(* Logix 5000 project; controller Google vendor 1 type 14 code 151 rev 31.11; software revision 31.00; part 2 of 6 *)

ADD_ON_INSTRUCTION Lift_Conv_Motor_Control   (* revision 1.0 *)
VAR_OUTPUT
   Motor_Data : SINT; {required}
END_VAR
VAR_INPUT
   Motor_FWD : BOOL; {required}
   Motor_REV : BOOL; {required}
   FWD_Speed : DINT; {required}
   REV_Speed : DINT; {required}
   Start_Delay : DINT; {required}
   Run_Permissive : DINT; {required}
END_VAR
VAR
   FWD_Delay : TIMER[4] := ([0].PRE := 500, [1].PRE := 500, [2].PRE := 500, [3].PRE := 500); {access None}
   REV_Delay : TIMER[4] := ([0].PRE := 500, [1].PRE := 500, [2].PRE := 500, [3].PRE := 500); {access None}
END_VAR

ROUTINE Logic   (* ladder *)
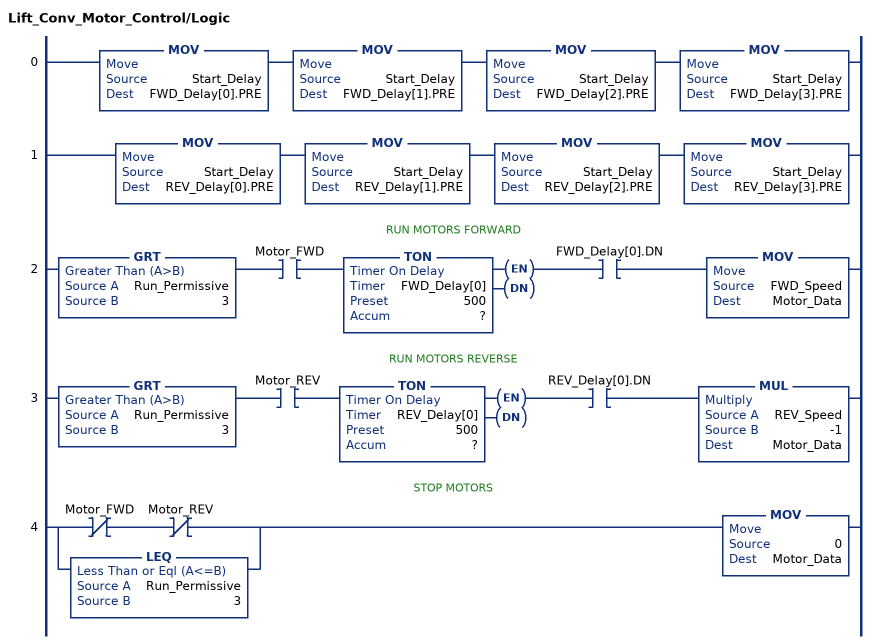
   0: MOV(Start_Delay,FWD_Delay[0].PRE)MOV(Start_Delay,FWD_Delay[1].PRE)MOV(Start_Delay,FWD_Delay[2].PRE)MOV(Start_Delay,FWD_Delay[3].PRE);
   1: MOV(Start_Delay,REV_Delay[0].PRE)MOV(Start_Delay,REV_Delay[1].PRE)MOV(Start_Delay,REV_Delay[2].PRE)MOV(Start_Delay,REV_Delay[3].PRE);
   // RUN MOTORS FORWARD
   2: GRT(Run_Permissive,3)XIC(Motor_FWD)TON(FWD_Delay[0],?,?)XIC(FWD_Delay[0].DN)MOV(FWD_Speed,Motor_Data);
   // RUN MOTORS REVERSE
   3: GRT(Run_Permissive,3)XIC(Motor_REV)TON(REV_Delay[0],?,?)XIC(REV_Delay[0].DN)MUL(REV_Speed,-1,Motor_Data);
   // STOP MOTORS
   4: [XIO(Motor_FWD) XIO(Motor_REV) ,LEQ(Run_Permissive,3) ]MOV(0,Motor_Data);
END_ROUTINE
END_ADD_ON_INSTRUCTION

ADD_ON_INSTRUCTION Lift_Conv_Sensor_Inputs   (* revision 1.0 *)
VAR_INPUT
   Data : SINT; {required}
END_VAR
VAR_OUTPUT
   Input_0 : BOOL; {access Read Only, required}
   Input_1 : BOOL; {access Read Only, required}
END_VAR

ROUTINE Logic   (* ladder *)
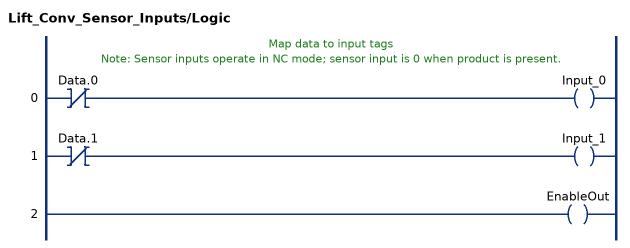
   // Map data to input tags
   // Note: Sensor inputs operate in NC mode; sensor input is 0 when product is present.
   0: XIO(Data.0)OTE(Input_0);
   1: XIO(Data.1)OTE(Input_1);
   2: OTE(EnableOut);
END_ROUTINE
END_ADD_ON_INSTRUCTION

ADD_ON_INSTRUCTION Lift_Zone_Data   (* revision 1.0 *)
VAR_IN_OUT
   Product_Name : STRING; {required}
   Product_Code : DINT; {required}
END_VAR
VAR_OUTPUT
   Occupied : BOOL; {access Read Only, visible}
END_VAR
VAR_INPUT
   Input_1 : BOOL; {required}
   Input_2 : BOOL; {required}
END_VAR
VAR_IN_OUT
   Upstream_ProdName : STRING; {required}
   Upstream_ProdCode : DINT; {required}
   Downstream_ProdName : STRING; {required}
   Downstream_ProdCode : DINT; {required}
END_VAR
VAR_INPUT
   FWD_Direction : BOOL; {required}
   REV_Direction : BOOL; {required}
END_VAR
VAR
   Blank_String : STRING; {access None}
   ONS : DINT; {access None}
   Occupied_Delay : TIMER := (PRE := 20); {access None}
   Unoccupied_Delay : TIMER := (PRE := 20); {access None}
END_VAR

ROUTINE Logic   (* ladder *)
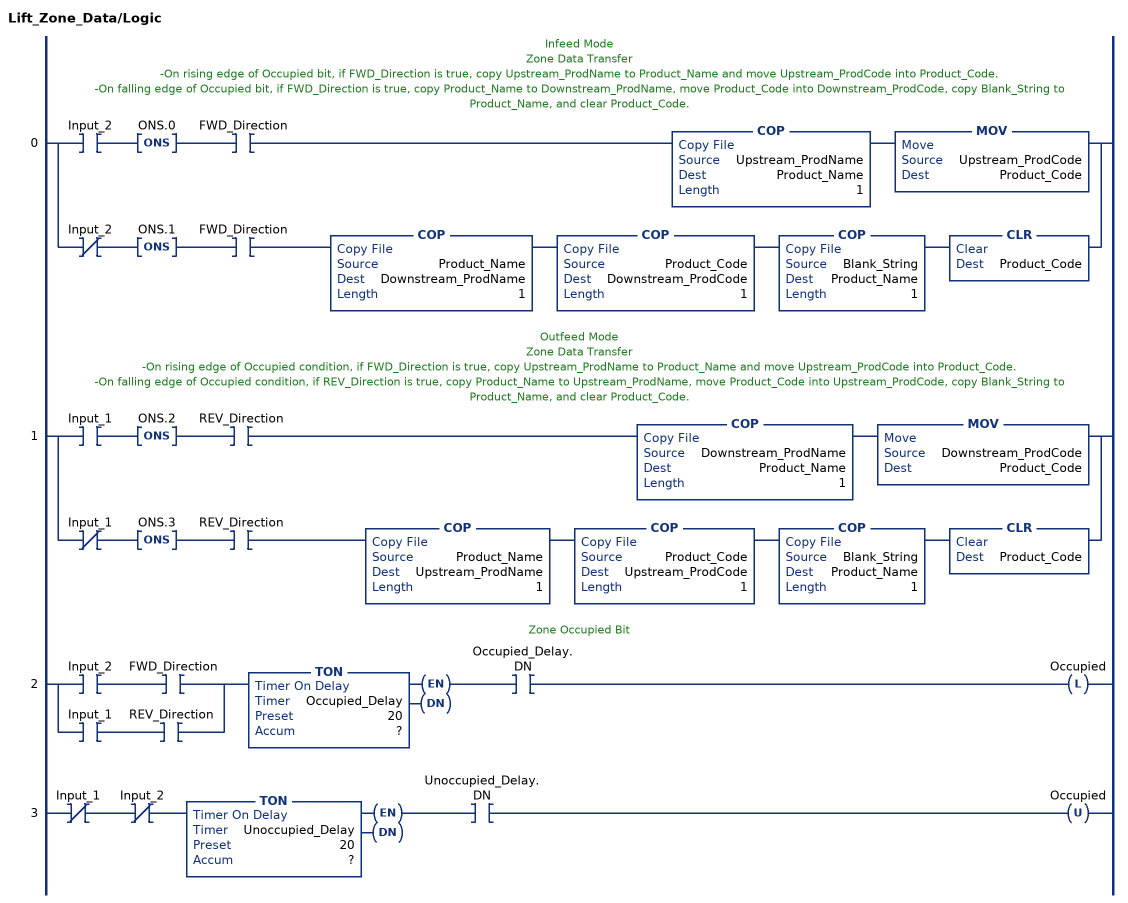
   // Infeed Mode
   // Zone Data Transfer
   // -On rising edge of Occupied bit, if FWD_Direction is true, copy Upstream_ProdName to Product_Name and move Upstream_ProdCode into Product_Code.
   // -On falling edge of Occupied bit, if FWD_Direction is true, copy Product_Name to Downstream_ProdName, move Product_Code into Downstream_ProdCode, copy Blank_String to Product_Name, and clear Product_Code.
   0: [XIC(Input_2) ONS(ONS.0) XIC(FWD_Direction) COP(Upstream_ProdName,Product_Name,1) MOV(Upstream_ProdCode,Product_Code) ,XIO(Input_2) ONS(ONS.1) XIC(FWD_Direction) COP(Product_Name,Downstream_ProdName,1) COP(Product_Code,Downstream_ProdCode,1) COP(Blank_String,Product_Name,1) CLR(Product_Code) ];
   // Outfeed Mode
   // Zone Data Transfer
   // -On rising edge of Occupied condition, if FWD_Direction is true, copy Upstream_ProdName to Product_Name and move Upstream_ProdCode into Product_Code.
   // -On falling edge of Occupied condition, if REV_Direction is true, copy Product_Name to Upstream_ProdName, move Product_Code into Upstream_ProdCode, copy Blank_String to Product_Name, and clear Product_Code.
   1: [XIC(Input_1) ONS(ONS.2) XIC(REV_Direction) COP(Downstream_ProdName,Product_Name,1) MOV(Downstream_ProdCode,Product_Code) ,XIO(Input_1) ONS(ONS.3) XIC(REV_Direction) COP(Product_Name,Upstream_ProdName,1) COP(Product_Code,Upstream_ProdCode,1) COP(Blank_String,Product_Name,1) CLR(Product_Code) ];
   // Zone Occupied Bit
   2: [XIC(Input_2) XIC(FWD_Direction) ,XIC(Input_1) XIC(REV_Direction) ]TON(Occupied_Delay,?,?)XIC(Occupied_Delay.DN)OTL(Occupied);
   3: XIO(Input_1)XIO(Input_2)TON(Unoccupied_Delay,?,?)XIC(Unoccupied_Delay.DN)OTU(Occupied);
END_ROUTINE
END_ADD_ON_INSTRUCTION

ADD_ON_INSTRUCTION Output_16_Bit   (* revision 1.0 *)
VAR_OUTPUT
   Output : BOOL; {access None}
   Data : INT; {required}
END_VAR
VAR_INPUT
   Output_0 : BOOL; {required}
   Output_1 : BOOL; {required}
   Output_2 : BOOL; {required}
   Output_3 : BOOL; {required}
   Output_4 : BOOL; {required}
   Output_5 : BOOL; {required}
   Output_6 : BOOL; {required}
   Output_7 : BOOL; {required}
   Output_8 : BOOL; {required}
   Output_9 : BOOL; {required}
   Output_10 : BOOL; {required}
   Output_11 : BOOL; {required}
   Output_12 : BOOL; {required}
   Output_13 : BOOL; {required}
   Output_14 : BOOL; {required}
   Output_15 : BOOL; {required}
   Test_Enable : BOOL; {required}
   Test_0 : BOOL; {required}
   Test_1 : BOOL; {required}
   Test_2 : BOOL; {required}
   Test_3 : BOOL; {required}
   Test_4 : BOOL; {required}
   Test_5 : BOOL; {required}
   Test_6 : BOOL; {required}
   Test_7 : BOOL; {required}
   Test_8 : BOOL; {required}
   Test_9 : BOOL; {required}
   Test_10 : BOOL; {required}
   Test_11 : BOOL; {required}
   Test_12 : BOOL; {required}
   Test_13 : BOOL; {required}
   Test_14 : BOOL; {required}
   Test_15 : BOOL; {required}
END_VAR
VAR
   ONS_Debounce : BOOL; {access None}
   Debounce_On_TMR : TIMER[16]; {access None}
   Debounce_Off_TMR : TIMER[16]; {access None}
END_VAR

ROUTINE Logic   (* ladder *)
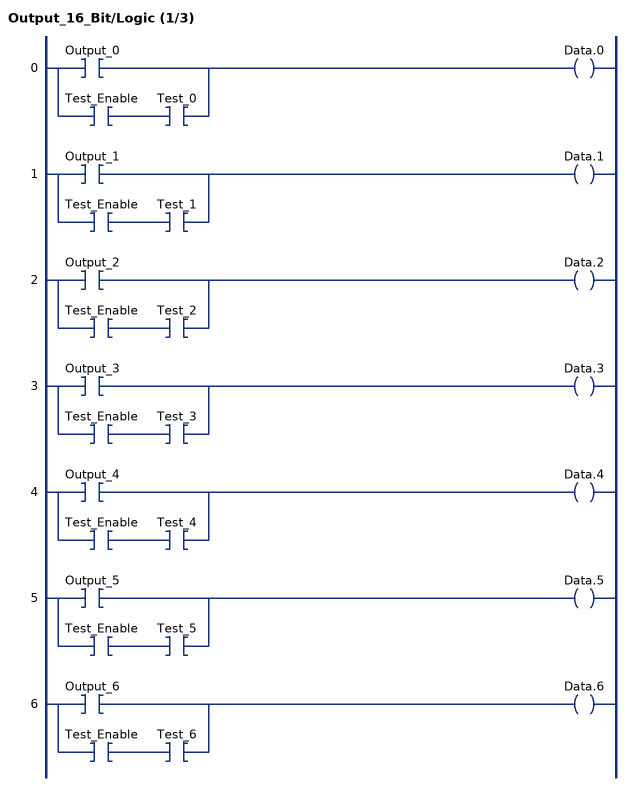
   0: [XIC(Output_0) ,XIC(Test_Enable) XIC(Test_0) ]OTE(Data.0);
   1: [XIC(Output_1) ,XIC(Test_Enable) XIC(Test_1) ]OTE(Data.1);
   2: [XIC(Output_2) ,XIC(Test_Enable) XIC(Test_2) ]OTE(Data.2);
   3: [XIC(Output_3) ,XIC(Test_Enable) XIC(Test_3) ]OTE(Data.3);
   4: [XIC(Output_4) ,XIC(Test_Enable) XIC(Test_4) ]OTE(Data.4);
   5: [XIC(Output_5) ,XIC(Test_Enable) XIC(Test_5) ]OTE(Data.5);
   6: [XIC(Output_6) ,XIC(Test_Enable) XIC(Test_6) ]OTE(Data.6);
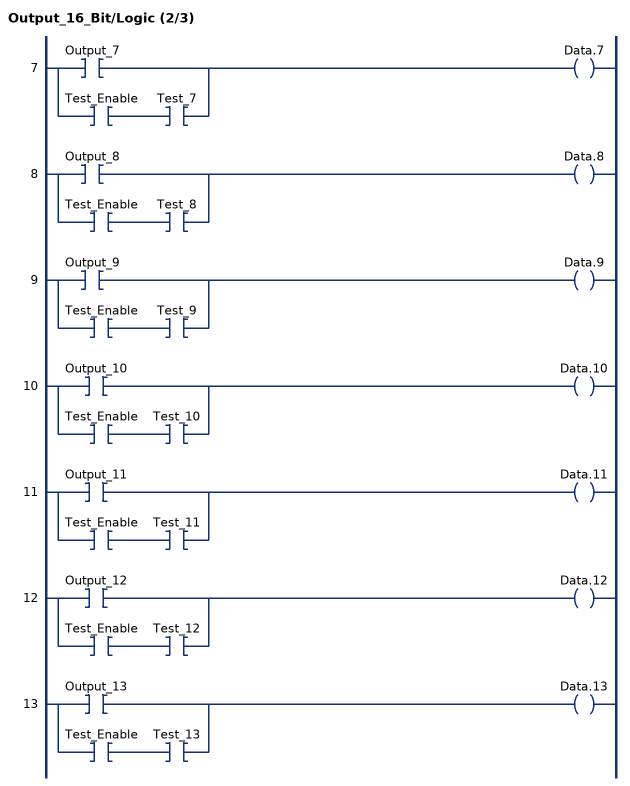
   7: [XIC(Output_7) ,XIC(Test_Enable) XIC(Test_7) ]OTE(Data.7);
   8: [XIC(Output_8) ,XIC(Test_Enable) XIC(Test_8) ]OTE(Data.8);
   9: [XIC(Output_9) ,XIC(Test_Enable) XIC(Test_9) ]OTE(Data.9);
   10: [XIC(Output_10) ,XIC(Test_Enable) XIC(Test_10) ]OTE(Data.10);
   11: [XIC(Output_11) ,XIC(Test_Enable) XIC(Test_11) ]OTE(Data.11);
   12: [XIC(Output_12) ,XIC(Test_Enable) XIC(Test_12) ]OTE(Data.12);
   13: [XIC(Output_13) ,XIC(Test_Enable) XIC(Test_13) ]OTE(Data.13);
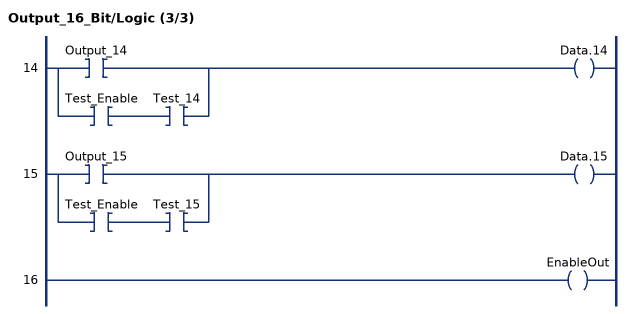
   14: [XIC(Output_14) ,XIC(Test_Enable) XIC(Test_14) ]OTE(Data.14);
   15: [XIC(Output_15) ,XIC(Test_Enable) XIC(Test_15) ]OTE(Data.15);
   16: OTE(EnableOut);
END_ROUTINE
END_ADD_ON_INSTRUCTION

ADD_ON_INSTRUCTION Pulser   (* revision 1.0 *)
VAR_INPUT
   On_Time : DINT; {required}
   Off_Time : DINT; {required}
END_VAR
VAR_OUTPUT
   Output : BOOL; {access Read Only}
END_VAR
VAR
   Pulse_ON_TMR : TIMER; {access None}
   Pulse_OFF_TMR : TIMER; {access None}
END_VAR

ROUTINE Logic   (* ladder *)
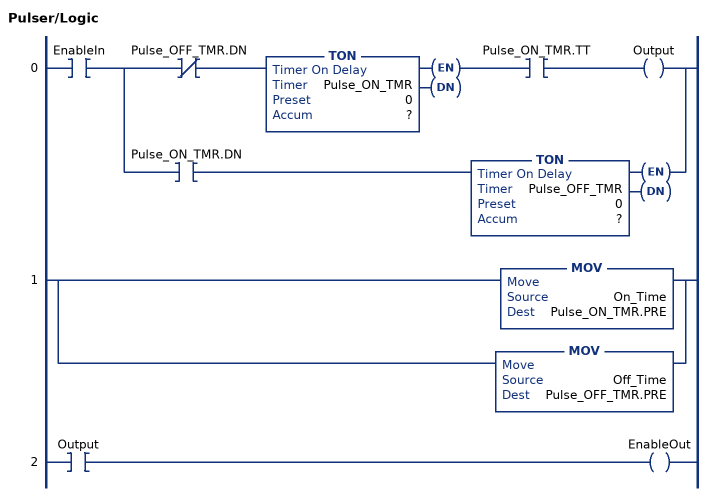
   0: XIC(EnableIn)[XIO(Pulse_OFF_TMR.DN) TON(Pulse_ON_TMR,?,?) XIC(Pulse_ON_TMR.TT) OTE(Output) ,XIC(Pulse_ON_TMR.DN) TON(Pulse_OFF_TMR,?,?) ];
   1: [MOV(On_Time,Pulse_ON_TMR.PRE) ,MOV(Off_Time,Pulse_OFF_TMR.PRE) ];
   2: XIC(Output)OTE(EnableOut);
END_ROUTINE
END_ADD_ON_INSTRUCTION

ADD_ON_INSTRUCTION Zone_Data   (* revision 1.0 *)
VAR_IN_OUT
   Product_Name : STRING; {required}
   Product_Code : DINT; {required}
END_VAR
VAR_OUTPUT
   Occupied : BOOL; {access Read Only, visible}
END_VAR
VAR_INPUT
   Input : BOOL; {required}
END_VAR
VAR_IN_OUT
   Upstream_ProdName : STRING; {required}
   Upstream_ProdCode : DINT; {required}
   Downstream_ProdName : STRING; {required}
   Downstream_ProdCode : DINT; {required}
END_VAR
VAR_INPUT
   FWD_Direction : BOOL; {required}
   REV_Direction : BOOL; {required}
END_VAR
VAR
   Blank_String : STRING; {access None}
   ONS : DINT; {access None}
   Occupied_Delay : TIMER := (PRE := 20); {access None}
END_VAR

ROUTINE Logic   (* ladder *)
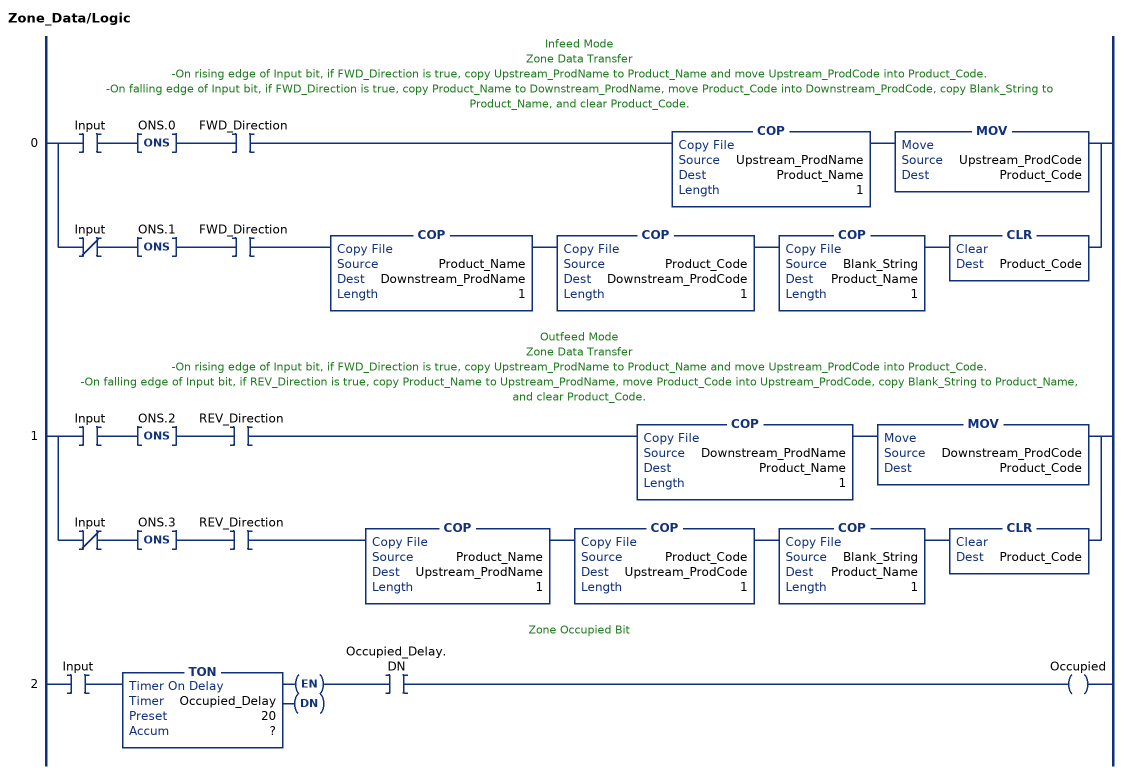
   // Infeed Mode
   // Zone Data Transfer
   // -On rising edge of Input bit, if FWD_Direction is true, copy Upstream_ProdName to Product_Name and move Upstream_ProdCode into Product_Code.
   // -On falling edge of Input bit, if FWD_Direction is true, copy Product_Name to Downstream_ProdName, move Product_Code into Downstream_ProdCode, copy Blank_String to Product_Name, and clear Product_Code.
   0: [XIC(Input) ONS(ONS.0) XIC(FWD_Direction) COP(Upstream_ProdName,Product_Name,1) MOV(Upstream_ProdCode,Product_Code) ,XIO(Input) ONS(ONS.1) XIC(FWD_Direction) COP(Product_Name,Downstream_ProdName,1) COP(Product_Code,Downstream_ProdCode,1) COP(Blank_String,Product_Name,1) CLR(Product_Code) ];
   // Outfeed Mode
   // Zone Data Transfer
   // -On rising edge of Input bit, if FWD_Direction is true, copy Upstream_ProdName to Product_Name and move Upstream_ProdCode into Product_Code.
   // -On falling edge of Input bit, if REV_Direction is true, copy Product_Name to Upstream_ProdName, move Product_Code into Upstream_ProdCode, copy Blank_String to Product_Name, and clear Product_Code.
   1: [XIC(Input) ONS(ONS.2) XIC(REV_Direction) COP(Downstream_ProdName,Product_Name,1) MOV(Downstream_ProdCode,Product_Code) ,XIO(Input) ONS(ONS.3) XIC(REV_Direction) COP(Product_Name,Upstream_ProdName,1) COP(Product_Code,Upstream_ProdCode,1) COP(Blank_String,Product_Name,1) CLR(Product_Code) ];
   // Zone Occupied Bit
   2: XIC(Input)TON(Occupied_Delay,?,?)XIC(Occupied_Delay.DN)OTE(Occupied);
END_ROUTINE
END_ADD_ON_INSTRUCTION

VAR_GLOBAL   (* controller tags *)
   Accum_Conv_Infeed : BOOL := 1;
   Accum_Conv_Outfeed : BOOL;
   Alarm : BOOL[64] := ([0] := 1);
   Alarm_Active : BOOL;
   Alarm_Delay : TIMER[32] := ([3].PRE := 100, [4].PRE := 5000, [5].PRE := 1000, [6].PRE := 1000, [7].PRE := 1000, [8].PRE := 1000, [9].PRE := 1000, [10].PRE := 1000, [11].PRE := 1000, [12].PRE := 1000, [13].PRE := 1000);
   Alarm_Horn : BOOL;
   Alarm_Pulser : Pulser := (On_Time := 500, Off_Time := 500);
   Alarm_Silence : BOOL;
   E_Stop_Pressed : BOOL;
   Elev_FWD_Delay : TIMER := (PRE := 100);
   Elev_REV_Delay : TIMER := (PRE := 100);
   Elev_Slow : BOOL;
   FaultResetDelay : TIMER := (PRE := 1000, ACC := 1001, EN := 1, DN := 1);
   GIB_MSG_CTRL : MESSAGE;
   HMI_Alarm_Silence : BOOL;
   HMI_AutoMode : BOOL := 1;
   HMI_Conv_FWD_Speed : DINT := 100;
   HMI_Conv_REV_Speed : DINT := 100;
   HMI_Conv_Start_Delay : DINT := 500;
   HMI_Infeed_Mode : BOOL := 1;
   HMI_Input1 : BOOL[32] := ([3] := 1, [4] := 1, [5] := 1);
   HMI_JogMode : BOOL;
   HMI_L2_Z1_Outfeed : BOOL;
   HMI_L2_Z2_Outfeed : BOOL;
   HMI_L2_Z3_Outfeed : BOOL;
   HMI_L2_Z4_Outfeed : BOOL;
   HMI_L3_Z1_Outfeed : BOOL;
   HMI_L3_Z2_Outfeed : BOOL;
   HMI_L3_Z3_Outfeed : BOOL;
   HMI_L3_Z4_Outfeed : BOOL;
   HMI_L4_Z1_Outfeed : BOOL;
   HMI_L4_Z2_Outfeed : BOOL;
   HMI_L4_Z3_Outfeed : BOOL;
   HMI_L4_Z4_Outfeed : BOOL;
   HMI_L5_Z1_Outfeed : BOOL;
   HMI_L5_Z2_Outfeed : BOOL;
   HMI_L5_Z3_Outfeed : BOOL;
   HMI_L5_Z4_Outfeed : BOOL;
   HMI_Lift_FullSpeed : DINT := 60;
   HMI_Lift_SlowSpeed : DINT := 20;
   HMI_Lift_Stop_Delay : DINT := 100;
   HMI_LiftJogDown : BOOL;
   HMI_LiftJogUp : BOOL;
   HMI_ManualMode : BOOL;
   HMI_Outfeed_Auto : BOOL;
   HMI_Outfeed_Batch : BOOL;
   HMI_Outfeed_Display : DINT;
   HMI_Outfeed_Mode : BOOL := 1;
   HMI_Outfeed_Single : BOOL := 1;
   HMI_Outfeed_Stop_Delay : DINT := 1000;
   HMI_Output1 : BOOL[32] := ([0] := 1, [4] := 1);
   HMI_OutputTest : BOOL[32];
   HMI_PB_Reset : BOOL;
   HMI_PB_Start : BOOL;
   HMI_PB_Stop : BOOL;
   HMI_System_Full : BOOL := 1;
   HMI_System_Mode : DINT;
   Infeed_Active : BOOL := 1;
   Infeed_Clear : BOOL;
   Infeed_Conv_Motors : Conveyor_Motor_Control := (FWD_Speed := 100, REV_Speed := 100, Start_Delay := 500, Run_Permissive := 4);
   Infeed_Conv_Sensors : Conv_Sensor_Inputs := (Data := 15, Infeed_Mode := 1, Outfeed_Stop_Delay := 1000);
   Infeed_Mode_Delay : TIMER := (PRE := 10000);
   Infeed_ModuleFaultCode : DINT;
   Infeed_Upstream_ProdCode : DINT;
   Infeed_Upstream_ProdName : STRING := ' ';
   Infeed_Z1_MinGapTimer : TIMER := (PRE := 3000);
   Infeed_Z1_ReleaseDelay : TIMER := (PRE := 2000);
   Infeed_Z3_MinGapTimer : TIMER := (PRE := 3000);
   Infeed_Zone1 : Zone_Data;
   Infeed_Zone1_2_ProdCode : DINT;
   Infeed_Zone1_2_ProdName : STRING;
   Infeed_Zone1_FWD : BOOL;
   Infeed_Zone1_PE : BOOL;
   Infeed_Zone1_ProdCode : DINT;
   Infeed_Zone1_ProdName : STRING;
   Infeed_Zone1_REV : BOOL;
   Infeed_Zone2 : Zone_Data;
   Infeed_Zone2_3_ProdCode : DINT;
   Infeed_Zone2_3_ProdName : STRING;
   Infeed_Zone2_FWD : BOOL;
   Infeed_Zone2_PE : BOOL;
   Infeed_Zone2_ProdCode : DINT;
   Infeed_Zone2_ProdName : STRING;
   Infeed_Zone2_REV : BOOL;
   Infeed_Zone3 : Zone_Data;
   Infeed_Zone3_4_ProdCode : DINT;
   Infeed_Zone3_4_ProdName : STRING;
   Infeed_Zone3_FWD : BOOL;
   Infeed_Zone3_PE : BOOL;
   Infeed_Zone3_ProdCode : DINT;
   Infeed_Zone3_ProdName : STRING;
   Infeed_Zone3_REV : BOOL;
   Infeed_Zone4 : Zone_Data;
   Infeed_Zone4_FWD : BOOL;
   Infeed_Zone4_PE : BOOL;
   Infeed_Zone4_ProdCode : DINT;
   Infeed_Zone4_ProdName : STRING;
   Infeed_Zone4_REV : BOOL;
   Infeed_Zone_Timeout : TIMER[8] := ([0].PRE := 5000, [0].ACC := 5000, [0].EN := 1, [0].DN := 1, [1].PRE := 10000, [2].PRE := 5000, [3].PRE := 10000, [4].PRE := 5000, [5].PRE := 5000, [6].PRE := 5000, [7].PRE := 5000);
   InfeedConv_Empty : BOOL;
   Inputs_1 : Input_16_Bit := (Data := 56, Input_3 := 1, Input_4 := 1, Input4_On_Debounce := 20, Input4_Off_Debounce := 20, Input_5 := 1, Input5_On_Debounce := 100, Input5_Off_Debounce := 20, Input6_On_Debounce := 20, Input6_Off_Debounce := 20, Input7_On_Debounce := 100, Input7_Off_Debounce := 20, Input8_On_Debounce := 20, Input8_Off_Debounce := 20, Input9_On_Debounce := 100, Input9_Off_Debounce := 20, Input10_On_Debounce := 20, Input10_Off_Debounce := 20, Input11_On_Debounce := 100, Input11_Off_Debounce := 20, Input12_On_Debounce := 100, Input12_Off_Debounce := 20, Input13_On_Debounce := 20, Input13_Off_Debounce := 20);
   L1_CearOutResetTimer : TIMER := (PRE := 5000);
   L1_Clear_Out : BOOL;
   L1_Conv_Motors : Conveyor_Motor_Control := (FWD_Speed := 100, REV_Speed := 100, Start_Delay := 500, Run_Permissive := 4);
   L1_Conv_Sensors : Conv_Sensor_Inputs := (Data := 15, Outfeed_Mode := 1, Outfeed_Stop_Delay := 1000);
   L1_Empty_Delay : TIMER := (PRE := 2000, ACC := 2000, EN := 1, DN := 1);
   L1_Full_Delay : TIMER := (PRE := 1000);
   L1_ModuleFaultCode : DINT;
   L1_Zone1 : Zone_Data;
   L1_Zone1_2_ProdCode : DINT;
   L1_Zone1_2_ProdName : STRING;
   L1_Zone1_FWD : BOOL;
   L1_Zone1_PE : BOOL;
   L1_Zone1_ProdCode : DINT;
   L1_Zone1_ProdName : STRING;
   L1_Zone1_REV : BOOL;
   L1_Zone2 : Zone_Data;
   L1_Zone2_3_ProdCode : DINT;
   L1_Zone2_3_ProdName : STRING;
   L1_Zone2_FWD : BOOL;
   L1_Zone2_PE : BOOL;
   L1_Zone2_ProdCode : DINT;
   L1_Zone2_ProdName : STRING;
   L1_Zone2_REV : BOOL;
   L1_Zone3 : Zone_Data;
   L1_Zone3_4_ProdCode : DINT;
   L1_Zone3_4_ProdName : STRING;
   L1_Zone3_FWD : BOOL;
   L1_Zone3_PE : BOOL;
   L1_Zone3_ProdCode : DINT;
   L1_Zone3_ProdName : STRING;
   L1_Zone3_REV : BOOL;
   L1_Zone4 : End_Zone_Data;
   L1_Zone4_FWD : BOOL;
   L1_Zone4_PE : BOOL;
   L1_Zone4_ProdCode : DINT;
   L1_Zone4_ProdName : STRING;
   L1_Zone4_REV : BOOL;
   L1_Zone_Timeout : TIMER[8] := ([0].PRE := 5000, [1].PRE := 10000, [2].PRE := 2000, [3].PRE := 6000, [4].PRE := 2000, [5].PRE := 5000, [6].PRE := 2000, [7].PRE := 5000);
   L2_Conv_Motors : Conveyor_Motor_Control := (FWD_Speed := 100, REV_Speed := 100, Start_Delay := 500, Run_Permissive := 4);
   L2_Conv_Sensors : Conv_Sensor_Inputs := (Input_0 := 1, Input_1 := 1, Input_2 := 1, Input_3 := 1, Infeed_Mode := 1, Outfeed_Stop_Delay := 1000);
   L2_Empty : BOOL;
   L2_Empty_Delay : TIMER := (PRE := 2000);
   L2_Full_Delay : TIMER := (PRE := 1000, ACC := 1001, EN := 1, DN := 1);
   L2_ModuleFaultCode : DINT;
   L2_Outfeed : BOOL;
   L2_Single_Outfeed : BOOL;
   L2_Z1_Outfeed : BOOL;
   L2_Z2_Outfeed : BOOL;
   L2_Z3_Outfeed : BOOL;
   L2_Z4_Outfeed : BOOL;
   L2_Zone1 : Zone_Data := (Occupied := 1, Input := 1);
   L2_Zone1_2_ProdCode : DINT;
   L2_Zone1_2_ProdName : STRING;
   L2_Zone1_FWD : BOOL;
   L2_Zone1_PE : BOOL := 1;
   L2_Zone1_ProdCode : DINT;
   L2_Zone1_ProdName : STRING;
   L2_Zone1_REV : BOOL;
   L2_Zone2 : Zone_Data := (Occupied := 1, Input := 1);
   L2_Zone2_3_ProdCode : DINT;
   L2_Zone2_3_ProdName : STRING;
   L2_Zone2_FWD : BOOL;
   L2_Zone2_PE : BOOL := 1;
   L2_Zone2_ProdCode : DINT;
   L2_Zone2_ProdName : STRING;
   L2_Zone2_REV : BOOL;
   L2_Zone3 : Zone_Data := (Occupied := 1, Input := 1);
   L2_Zone3_4_ProdCode : DINT;
   L2_Zone3_4_ProdName : STRING := ' ';
   L2_Zone3_FWD : BOOL;
   L2_Zone3_PE : BOOL := 1;
   L2_Zone3_ProdCode : DINT;
   L2_Zone3_ProdName : STRING;
   L2_Zone3_REV : BOOL;
   L2_Zone4 : End_Zone_Data := (Occupied := 1, Input := 1);
   L2_Zone4_FWD : BOOL;
   L2_Zone4_PE : BOOL := 1;
   L2_Zone4_ProdCode : DINT;
   L2_Zone4_ProdName : STRING := ' ';
   L2_Zone4_REV : BOOL;
   L2_Zone_Timeout : TIMER[8] := ([0].PRE := 5000, [1].PRE := 10000, [2].PRE := 5000, [3].PRE := 5000, [4].PRE := 5000, [5].PRE := 5000, [6].PRE := 5000, [7].PRE := 5000);
   L3_Conv_Motors : Conveyor_Motor_Control := (FWD_Speed := 100, REV_Speed := 100, Start_Delay := 500, Run_Permissive := 4);
   L3_Conv_Sensors : Conv_Sensor_Inputs := (Input_0 := 1, Input_1 := 1, Input_2 := 1, Input_3 := 1, Infeed_Mode := 1, Outfeed_Stop_Delay := 1000);
   L3_Empty : BOOL;
   L3_Empty_Delay : TIMER := (PRE := 2000);
   L3_Full_Delay : TIMER := (PRE := 1000, ACC := 1000, EN := 1, DN := 1);
   L3_ModuleFaultCode : DINT;
   L3_Outfeed : BOOL;
   L3_Single_Outfeed : BOOL;
   L3_Z1_Outfeed : BOOL;
   L3_Z2_Outfeed : BOOL;
   L3_Z3_Outfeed : BOOL;
   L3_Z4_Outfeed : BOOL;
   L3_Zone1 : Zone_Data := (Occupied := 1, Input := 1);
   L3_Zone1_2_ProdCode : DINT;
   L3_Zone1_2_ProdName : STRING;
   L3_Zone1_FWD : BOOL;
   L3_Zone1_PE : BOOL := 1;
   L3_Zone1_ProdCode : DINT;
   L3_Zone1_ProdName : STRING;
   L3_Zone1_REV : BOOL;
   L3_Zone2 : Zone_Data := (Occupied := 1, Input := 1);
   L3_Zone2_3_ProdCode : DINT;
   L3_Zone2_3_ProdName : STRING;
   L3_Zone2_FWD : BOOL;
   L3_Zone2_PE : BOOL := 1;
   L3_Zone2_ProdCode : DINT;
   L3_Zone2_ProdName : STRING;
   L3_Zone2_REV : BOOL;
   L3_Zone3 : Zone_Data := (Occupied := 1, Input := 1);
   L3_Zone3_4_ProdCode : DINT;
   L3_Zone3_4_ProdName : STRING := ' ';
   L3_Zone3_FWD : BOOL;
   L3_Zone3_PE : BOOL := 1;
   L3_Zone3_ProdCode : DINT;
   L3_Zone3_ProdName : STRING;
   L3_Zone3_REV : BOOL;
   L3_Zone4 : End_Zone_Data := (Occupied := 1, Input := 1);
   L3_Zone4_FWD : BOOL;
   L3_Zone4_PE : BOOL := 1;
   L3_Zone4_ProdCode : DINT;
   L3_Zone4_ProdName : STRING := ' ';
   L3_Zone4_REV : BOOL;
   L3_Zone_Timeout : TIMER[8] := ([0].PRE := 5000, [1].PRE := 10000, [2].PRE := 5000, [3].PRE := 5000, [4].PRE := 5000, [5].PRE := 5000, [6].PRE := 5000, [7].PRE := 5000);
   L4_Conv_Motors : Conveyor_Motor_Control := (FWD_Speed := 100, REV_Speed := 100, Start_Delay := 500, Run_Permissive := 4);
   L4_Conv_Sensors : Conv_Sensor_Inputs := (Input_0 := 1, Input_1 := 1, Input_2 := 1, Input_3 := 1, Infeed_Mode := 1, Outfeed_Stop_Delay := 1000);
   L4_Empty : BOOL;
   L4_Empty_Delay : TIMER := (PRE := 2000);
   L4_Full_Delay : TIMER := (PRE := 1000, ACC := 1000, EN := 1, DN := 1);
   L4_ModuleFaultCode : DINT;
   L4_Outfeed : BOOL;
   L4_Single_Outfeed : BOOL;
   L4_Z1_Outfeed : BOOL;
   L4_Z2_Outfeed : BOOL;
   L4_Z3_Outfeed : BOOL;
   L4_Z4_Outfeed : BOOL;
   L4_Zone1 : Zone_Data := (Occupied := 1, Input := 1);
   L4_Zone1_2_ProdCode : DINT;
   L4_Zone1_2_ProdName : STRING;
   L4_Zone1_FWD : BOOL;
   L4_Zone1_PE : BOOL := 1;
   L4_Zone1_ProdCode : DINT;
   L4_Zone1_ProdName : STRING;
   L4_Zone1_REV : BOOL;
   L4_Zone2 : Zone_Data := (Occupied := 1, Input := 1);
   L4_Zone2_3_ProdCode : DINT;
   L4_Zone2_3_ProdName : STRING;
   L4_Zone2_FWD : BOOL;
   L4_Zone2_PE : BOOL := 1;
   L4_Zone2_ProdCode : DINT;
   L4_Zone2_ProdName : STRING;
   L4_Zone2_REV : BOOL;
   L4_Zone3 : Zone_Data := (Occupied := 1, Input := 1);
   L4_Zone3_4_ProdCode : DINT;
   L4_Zone3_4_ProdName : STRING;
   L4_Zone3_FWD : BOOL;
   L4_Zone3_PE : BOOL := 1;
   L4_Zone3_ProdCode : DINT;
   L4_Zone3_ProdName : STRING;
   L4_Zone3_REV : BOOL;
   L4_Zone4 : End_Zone_Data := (Occupied := 1, Input := 1);
   L4_Zone4_FWD : BOOL;
   L4_Zone4_PE : BOOL := 1;
   L4_Zone4_ProdCode : DINT;
   L4_Zone4_ProdName : STRING;
   L4_Zone4_REV : BOOL;
   L4_Zone_Timeout : TIMER[8] := ([0].PRE := 5000, [1].PRE := 10000, [2].PRE := 5000, [3].PRE := 5000, [4].PRE := 5000, [5].PRE := 5000, [6].PRE := 5000, [7].PRE := 5000);
   L5_Conv_Motors : Conveyor_Motor_Control := (FWD_Speed := 100, REV_Speed := 100, Start_Delay := 500, Run_Permissive := 4);
   L5_Conv_Sensors : Conv_Sensor_Inputs := (Input_0 := 1, Input_1 := 1, Input_2 := 1, Input_3 := 1, Infeed_Mode := 1, Outfeed_Stop_Delay := 1000);
   L5_Empty : BOOL;
   L5_Empty_Delay : TIMER := (PRE := 2000);
   L5_Full_Delay : TIMER := (PRE := 1000, ACC := 1000, EN := 1, DN := 1);
   L5_ModuleFaultCode : DINT;
   L5_Outfeed : BOOL;
   L5_Single_Outfeed : BOOL;
   L5_Z1_Outfeed : BOOL;
   L5_Z2_Outfeed : BOOL;
   L5_Z3_Outfeed : BOOL;
   L5_Z4_Outfeed : BOOL;
   L5_Zone1 : Zone_Data := (Occupied := 1, Input := 1);
   L5_Zone1_2_ProdCode : DINT;
   L5_Zone1_2_ProdName : STRING;
   L5_Zone1_FWD : BOOL;
   L5_Zone1_PE : BOOL := 1;
   L5_Zone1_ProdCode : DINT;
   L5_Zone1_ProdName : STRING;
   L5_Zone1_REV : BOOL;
   L5_Zone2 : Zone_Data := (Occupied := 1, Input := 1);
   L5_Zone2_3_ProdCode : DINT;
   L5_Zone2_3_ProdName : STRING;
   L5_Zone2_FWD : BOOL;
   L5_Zone2_PE : BOOL := 1;
   L5_Zone2_ProdCode : DINT;
   L5_Zone2_ProdName : STRING;
   L5_Zone2_REV : BOOL;
   L5_Zone3 : Zone_Data := (Occupied := 1, Input := 1);
   L5_Zone3_4_ProdCode : DINT;
   L5_Zone3_4_ProdName : STRING;
   L5_Zone3_FWD : BOOL;
   L5_Zone3_PE : BOOL := 1;
   L5_Zone3_ProdCode : DINT;
   L5_Zone3_ProdName : STRING;
   L5_Zone3_REV : BOOL;
   L5_Zone4 : End_Zone_Data := (Occupied := 1, Input := 1);
   L5_Zone4_FWD : BOOL;
   L5_Zone4_PE : BOOL := 1;
   L5_Zone4_ProdCode : DINT;
   L5_Zone4_ProdName : STRING;
   L5_Zone4_REV : BOOL;
   L5_Zone_Timeout : TIMER[8] := ([0].PRE := 5000, [1].PRE := 10000, [2].PRE := 2000, [3].PRE := 5000, [4].PRE := 2000, [5].PRE := 5000, [6].PRE := 2000, [7].PRE := 5000);
   Level_1_Empty : BOOL := 1;
   Level_1_Full : BOOL;
   Level_2_Empty : BOOL;
   Level_2_Full : BOOL := 1;
   Level_3_Empty : BOOL;
   Level_3_Full : BOOL := 1;
   Level_4_Empty : BOOL;
   Level_4_Full : BOOL := 1;
   Level_5_Empty : BOOL;
   Level_5_Full : BOOL := 1;
   Lift_Alarm : BOOL;
   Lift_Ascend : BOOL;
   Lift_Conv_Motor : Lift_Conv_Motor_Control := (FWD_Speed := 100, REV_Speed := 100, Start_Delay := 500, Run_Permissive := 4);
   Lift_Conv_PE1 : BOOL;
   Lift_Conv_PE2 : BOOL;
   Lift_Conv_Sensors : Lift_Conv_Sensor_Inputs := (Data := 3);
   Lift_Current_Level : DINT := 1;
   Lift_Cycle_Counter : COUNTER := (ACC := 1297, CU := 1, DN := 1);
   Lift_Descend : BOOL;
   Lift_FullSpeed : DINT := 6000;
   Lift_L1_Slow_Prox : BOOL := 1;
   Lift_L1_Stop_Prox : BOOL := 1;
   Lift_L2_Slow_Prox : BOOL;
   Lift_L2_Stop_Prox : BOOL;
   Lift_L3_Slow_Prox : BOOL;
   Lift_L3_Stop_Prox : BOOL;
   Lift_L4_Slow_Prox : BOOL;
   Lift_L4_Stop_Prox : BOOL;
   Lift_L5_Slow_Prox : BOOL;
   Lift_L5_Stop_Prox : BOOL;
   Lift_ModuleFaultCode : DINT;
   Lift_Required_Level : DINT := 1;
   Lift_SlowSpeed : DINT := 2000;
   Lift_Zone : Lift_Zone_Data;
   Lift_Zone_ProdCode : DINT;
   Lift_Zone_ProdName : STRING;
   Lift_Zone_Timeout : TIMER[2] := ([0].PRE := 3000, [1].PRE := 3000);
   LiftConv_Empty : BOOL;
   LiftZone_FWD : BOOL;
   LiftZone_REV : BOOL;
   LiftZoneDownstream_ProdCode : DINT;
   LiftZoneDownstream_ProdName : STRING;
   LiftZoneFWD_ResetTimer : TIMER := (PRE := 10);
   LiftZoneREV_ResetTimer : TIMER := (PRE := 10);
   LiftZoneUpstream_ProdCode : DINT;
   LiftZoneUpstream_ProdName : STRING;
   Manual_Mode_Active : BOOL;
   MCR_DelayActive : BOOL;
   MCR_Enable : BOOL := 1;
   MCR_EnableDelay : TIMER := (PRE := 5000);
   MCR_Status : BOOL;
   Motion_Complete : BOOL := 1;
   MotionStoppedTimer : TIMER := (PRE := 10000, ACC := 10000, EN := 1, DN := 1);
   ONS : DINT[6] := ([1] := 1644167168, [2] := 3, [3] := 1);
   Outfeed_Active : BOOL;
   Outfeed_Automatic : BOOL;
   Outfeed_Batch : BOOL;
   Outfeed_In_Process : BOOL;
   Outfeed_Mode_Delay : TIMER := (PRE := 10000, ACC := 10000, EN := 1, DN := 1);
   Outfeed_Single : BOOL;
   Outputs_1 : Output_16_Bit := (Data := 17, Output_0 := 1, Output_4 := 1);
   PS10017_DC_OK : BOOL := 1;
   Ready_Pulser : Pulser := (On_Time := 500, Off_Time := 500);
   Request_LSTleft_Trigger : BOOL := 1;
   Request_LSTright_Trigger : BOOL := 1;
   Safety_OK : BOOL := 1;
   Safety_OK_Delay : TIMER := (PRE := 15000, ACC := 15001, EN := 1, DN := 1);
   Safety_Relay_Status : BOOL;
   Sort_Number : DINT;
   Sorting_Active : BOOL;
   Sorting_Inactive : BOOL := 1;
   Spare_Input : BOOL;
   Spare_Output : BOOL;
   Stacklight_Amber : BOOL;
   Stacklight_Audible : BOOL;
   Stacklight_Green : BOOL := 1;
   Stacklight_Red : BOOL;
   Starting_Horn : BOOL;
   Starting_Pulser : Pulser := (On_Time := 800, Off_Time := 800, Output := 1);
   Stopping_Pulser : Pulser := (On_Time := 1000, Off_Time := 1000);
   System : State := (Resetting := 1, Ready := 2, Starting := 3, Running := 4, Stopping := 5); {constant}
   System_Mode_Change : BOOL;
   System_State : DINT := 4;
   SystemStartDelay : TIMER := (PRE := 5000);
   Test : DINT := 1;
   Test_Timer : TIMER[10] := ([0].PRE := 5000, [1].PRE := 500, [2].PRE := 500, [3].PRE := 500, [4].PRE := 500, [5].PRE := 50, [6].PRE := 50, [7].PRE := 50);
END_VAR

PROGRAM IPC_Program   (* main routine MainRoutine *)
VAR
   CsharpTag : BOOL;
   IPC_Control_Active : BOOL;
END_VAR

ROUTINE C01_Comms   (* ladder *)
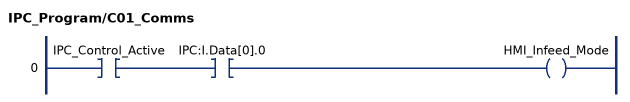
   0: XIC(IPC_Control_Active)XIC(IPC:I.Data[0].0)OTE(HMI_Infeed_Mode);
END_ROUTINE

ROUTINE MainRoutine   (* ladder *)
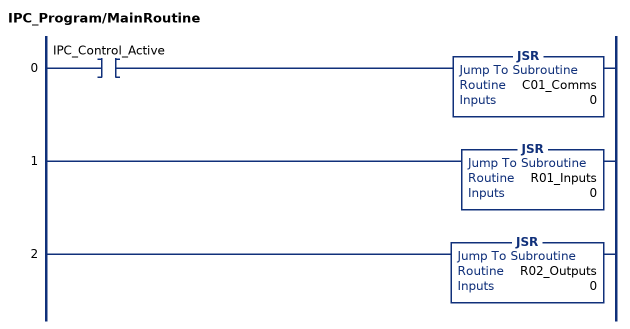
   0: XIC(IPC_Control_Active)JSR(C01_Comms,0);
   1: JSR(R01_Inputs,0);
   2: JSR(R02_Outputs,0);
END_ROUTINE

ROUTINE R01_Inputs   (* ladder *)
   0: NOP();
END_ROUTINE

ROUTINE R02_Outputs   (* ladder *)
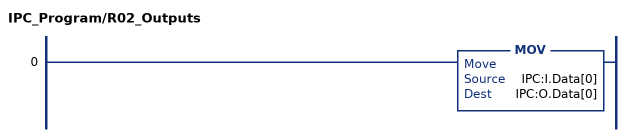
   0: MOV(IPC:I.Data[0],IPC:O.Data[0]);
END_ROUTINE
END_PROGRAM

PROGRAM MainProgram   (* main routine MainRoutine *)

ROUTINE C01_Comms   (* ladder *)
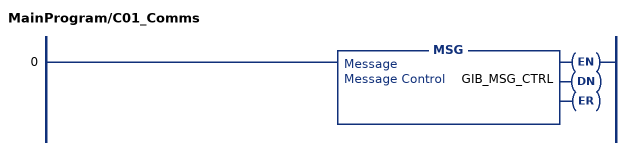
   0: MSG(GIB_MSG_CTRL);
END_ROUTINE

ROUTINE MainRoutine   (* ladder *)
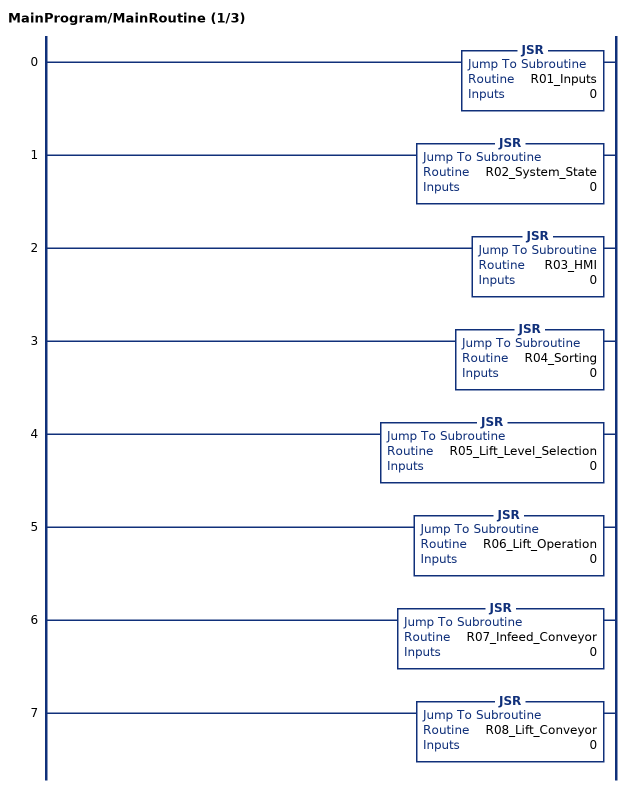
   0: JSR(R01_Inputs,0);
   1: JSR(R02_System_State,0);
   2: JSR(R03_HMI,0);
   3: JSR(R04_Sorting,0);
   4: JSR(R05_Lift_Level_Selection,0);
   5: JSR(R06_Lift_Operation,0);
   6: JSR(R07_Infeed_Conveyor,0);
   7: JSR(R08_Lift_Conveyor,0);
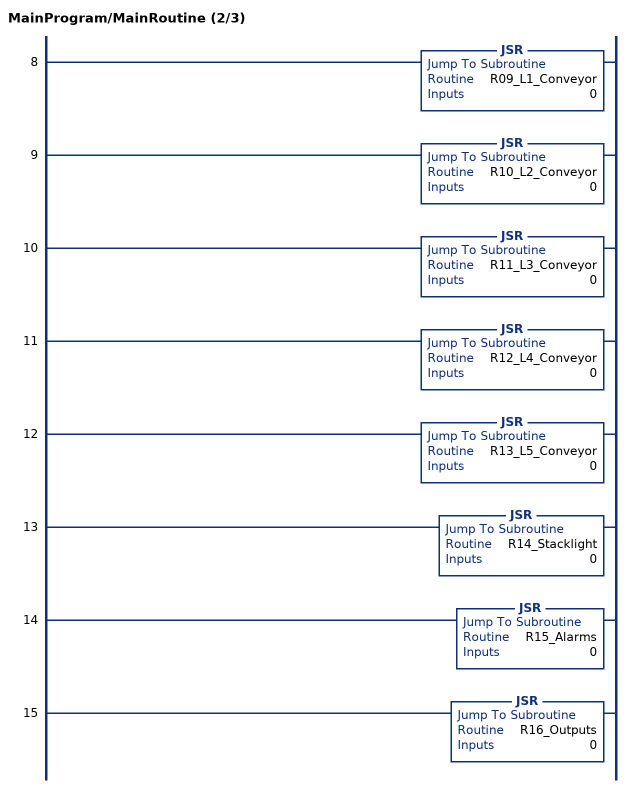
   8: JSR(R09_L1_Conveyor,0);
   9: JSR(R10_L2_Conveyor,0);
   10: JSR(R11_L3_Conveyor,0);
   11: JSR(R12_L4_Conveyor,0);
   12: JSR(R13_L5_Conveyor,0);
   13: JSR(R14_Stacklight,0);
   14: JSR(R15_Alarms,0);
   15: JSR(R16_Outputs,0);
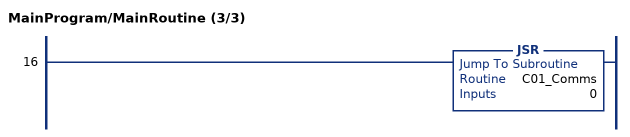
   16: JSR(C01_Comms,0);
END_ROUTINE

ROUTINE R01_Inputs   (* ladder *)
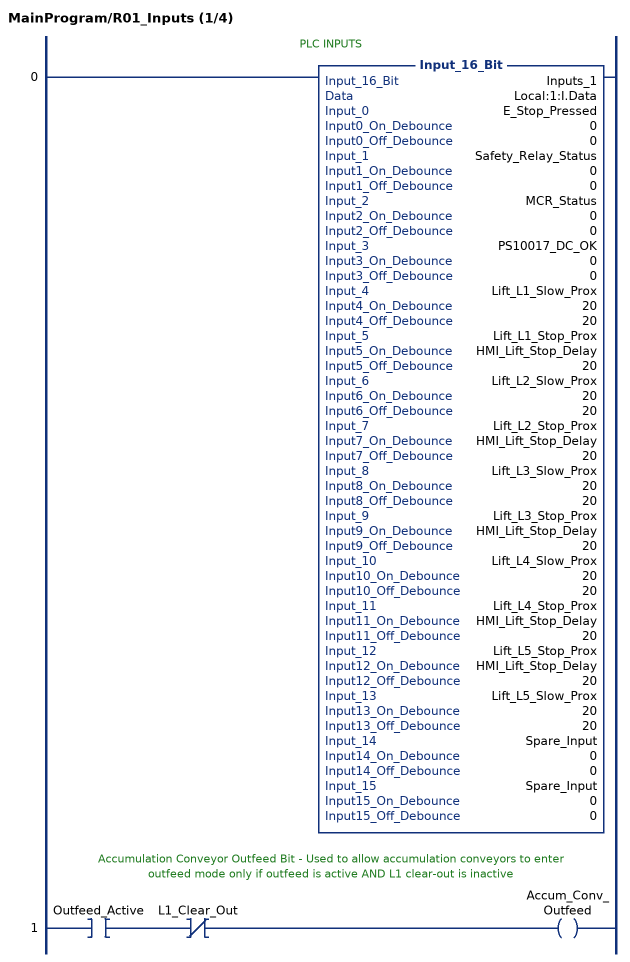
   // PLC INPUTS
   0: Input_16_Bit(Inputs_1,Local:1:I.Data,E_Stop_Pressed,0,0,Safety_Relay_Status,0,0,MCR_Status,0,0,PS10017_DC_OK,0,0,Lift_L1_Slow_Prox,20,20,Lift_L1_Stop_Prox,HMI_Lift_Stop_Delay,20,Lift_L2_Slow_Prox,20,20,Lift_L2_Stop_Prox,HMI_Lift_Stop_Delay,20,Lift_L3_Slow_Prox,20,20,Lift_L3_Stop_Prox,HMI_Lift_Stop_Delay,20,Lift_L4_Slow_Prox,20,20,Lift_L4_Stop_Prox,HMI_Lift_Stop_Delay,20,Lift_L5_Stop_Prox,HMI_Lift_Stop_Delay,20,Lift_L5_Slow_Prox,20,20,Spare_Input,0,0,Spare_Input,0,0);
   // Accumulation Conveyor Outfeed Bit - Used to allow accumulation conveyors to enter outfeed mode only if outfeed is active AND L1 clear-out is inactive
   1: XIC(Outfeed_Active)XIO(L1_Clear_Out)OTE(Accum_Conv_Outfeed);
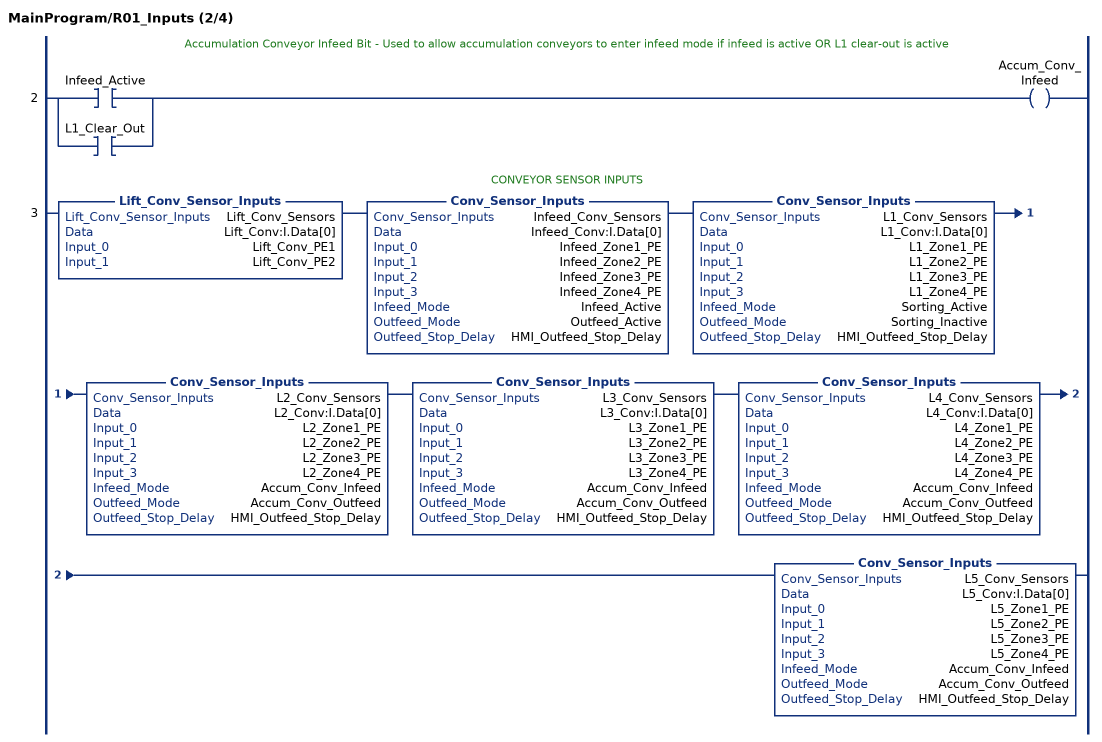
   // Accumulation Conveyor Infeed Bit - Used to allow accumulation conveyors to enter infeed mode if infeed is active OR L1 clear-out is active
   2: [XIC(Infeed_Active) ,XIC(L1_Clear_Out) ]OTE(Accum_Conv_Infeed);
   // CONVEYOR SENSOR INPUTS
   3: Lift_Conv_Sensor_Inputs(Lift_Conv_Sensors,Lift_Conv:I.Data[0],Lift_Conv_PE1,Lift_Conv_PE2)Conv_Sensor_Inputs(Infeed_Conv_Sensors,Infeed_Conv:I.Data[0],Infeed_Zone1_PE,Infeed_Zone2_PE,Infeed_Zone3_PE,Infeed_Zone4_PE,Infeed_Active,Outfeed_Active,HMI_Outfeed_Stop_Delay)Conv_Sensor_Inputs(L1_Conv_Sensors,L1_Conv:I.Data[0],L1_Zone1_PE,L1_Zone2_PE,L1_Zone3_PE,L1_Zone4_PE,Sorting_Active,Sorting_Inactive,HMI_Outfeed_Stop_Delay)Conv_Sensor_Inputs(L2_Conv_Sensors,L2_Conv:I.Data[0],L2_Zone1_PE,L2_Zone2_PE,L2_Zone3_PE,L2_Zone4_PE,Accum_Conv_Infeed,Accum_Conv_Outfeed,HMI_Outfeed_Stop_Delay)Conv_Sensor_Inputs(L3_Conv_Sensors,L3_Conv:I.Data[0],L3_Zone1_PE,L3_Zone2_PE,L3_Zone3_PE,L3_Zone4_PE,Accum_Conv_Infeed,Accum_Conv_Outfeed,HMI_Outfeed_Stop_Delay)Conv_Sensor_Inputs(L4_Conv_Sensors,L4_Conv:I.Data[0],L4_Zone1_PE,L4_Zone2_PE,L4_Zone3_PE,L4_Zone4_PE,Accum_Conv_Infeed,Accum_Conv_Outfeed,HMI_Outfeed_Stop_Delay)Conv_Sensor_Inputs(L5_Conv_Sensors,L5_Conv:I.Data[0],L5_Zone1_PE,L5_Zone2_PE,L5_Zone3_PE,L5_Zone4_PE,Accum_Conv_Infeed,Accum_Conv_Outfeed,HMI_Outfeed_Stop_Delay);
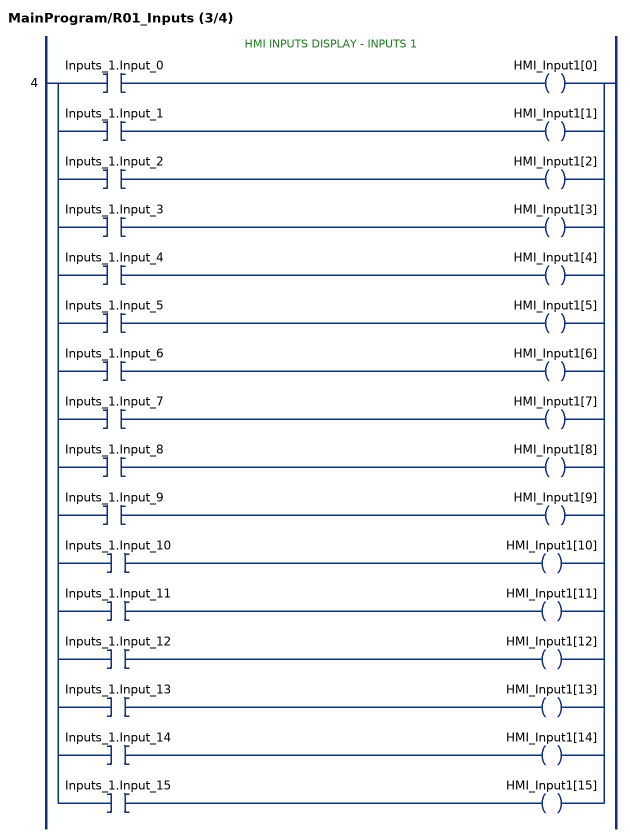
   // HMI INPUTS DISPLAY - INPUTS 1
   4: [XIC(Inputs_1.Input_0) OTE(HMI_Input1[0]) ,XIC(Inputs_1.Input_1) OTE(HMI_Input1[1]) ,XIC(Inputs_1.Input_2) OTE(HMI_Input1[2]) ,XIC(Inputs_1.Input_3) OTE(HMI_Input1[3]) ,XIC(Inputs_1.Input_4) OTE(HMI_Input1[4]) ,XIC(Inputs_1.Input_5) OTE(HMI_Input1[5]) ,XIC(Inputs_1.Input_6) OTE(HMI_Input1[6]) ,XIC(Inputs_1.Input_7) OTE(HMI_Input1[7]) ,XIC(Inputs_1.Input_8) OTE(HMI_Input1[8]) ,XIC(Inputs_1.Input_9) OTE(HMI_Input1[9]) ,XIC(Inputs_1.Input_10) OTE(HMI_Input1[10]) ,XIC(Inputs_1.Input_11) OTE(HMI_Input1[11]) ,XIC(Inputs_1.Input_12) OTE(HMI_Input1[12]) ,XIC(Inputs_1.Input_13) OTE(HMI_Input1[13]) ,XIC(Inputs_1.Input_14) OTE(HMI_Input1[14]) ,XIC(Inputs_1.Input_15) OTE(HMI_Input1[15]) ];
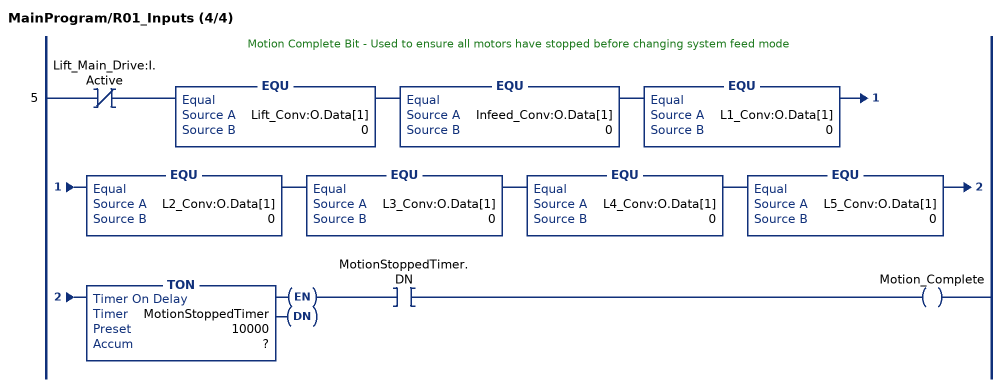
   // Motion Complete Bit - Used to ensure all motors have stopped before changing system feed mode
   5: XIO(Lift_Main_Drive:I.Active)EQU(Lift_Conv:O.Data[1],0)EQU(Infeed_Conv:O.Data[1],0)EQU(L1_Conv:O.Data[1],0)EQU(L2_Conv:O.Data[1],0)EQU(L3_Conv:O.Data[1],0)EQU(L4_Conv:O.Data[1],0)EQU(L5_Conv:O.Data[1],0)TON(MotionStoppedTimer,?,?)XIC(MotionStoppedTimer.DN)OTE(Motion_Complete);
END_ROUTINE
